// TIA Portal V19 export
TYPE "LEXCHANGETRAY_typeRoller_toLogisticsFeedback_B2"
// stored: Access Published
   STRUCT
      inFeedEnabled : Bool;   // 允许进料
      outFeeding : Bool;   // 进料中
   END_STRUCT;
END_TYPE
